// TIA Portal V20 export
TYPE "UDT_Service_Information"
   STRUCT
      state { ExternalWritable := 'False'} : DWord;   // S88 State
      lastState { ExternalWritable := 'False'} : DWord;   // S88 last State
      readyToComplete { ExternalWritable := 'False'} : Bool;   // Ready to complete active
      startTime { ExternalWritable := 'False'} : DTL;   // Start time of control sequence
      endTime { ExternalWritable := 'False'} : DTL;   // End time of control sequence
   END_STRUCT;
END_TYPE
